SUBAPPLICATION Uebung_035a_AX (* Lauflicht 4 reine Zeitsteuerung (Adapter Version) *)
  (* Standard: 61499-2; Description: Copyright (c) 2026 Meisterschulen am Ostbahnhof This program and the accompanying materials are made available under the terms of the Eclipse Public License 2.0 which is available at https://www.eclipse.org/legal/epl-2.0/ SPDX-License-Identifier: EPL-2.0 *)
  (* Version 1.0, 2026-07-05, Franz Höpfinger, Meisterschulen am Ostbahnhof, generated solution *)
  PACKAGE Uebungen;
  IMPORT Uebungen::const::UT::DefaultPool::OutputNumber_N1;
  IMPORT logiBUS::io::DI::logiBUS_DI::Input_I1;
  IMPORT logiBUS::io::DI::logiBUS_DI::Input_I2;
  IMPORT logiBUS::io::DI::logiBUS_DI::Input_I3;
  IMPORT logiBUS::io::DI::logiBUS_DI::Input_I4;
  IMPORT logiBUS::io::DI::logiBUS_DI_Events::BUTTON_SINGLE_CLICK;
  IMPORT logiBUS::io::DQ::logiBUS_DO::Output_Q1;
  IMPORT logiBUS::io::DQ::logiBUS_DO::Output_Q2;
  IMPORT logiBUS::io::DQ::logiBUS_DO::Output_Q3;
  IMPORT logiBUS::io::DQ::logiBUS_DO::Output_Q4;
  IMPORT logiBUS::utils::sequence::const::sequence::NO_TIME;
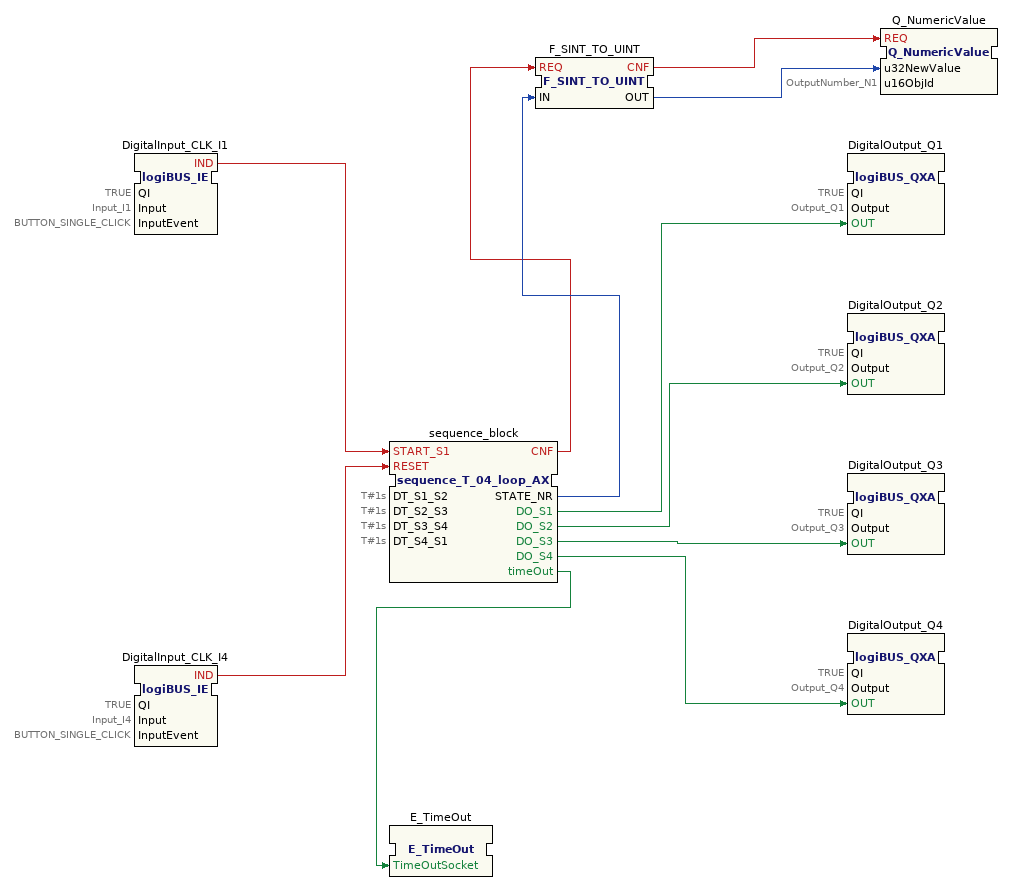
  FBS
    DigitalOutput_Q1 : logiBUS::io::DQ::logiBUS_QXA(QI := TRUE, Output := Output_Q1);
    DigitalOutput_Q2 : logiBUS::io::DQ::logiBUS_QXA(QI := TRUE, Output := Output_Q2);
    DigitalOutput_Q3 : logiBUS::io::DQ::logiBUS_QXA(QI := TRUE, Output := Output_Q3);
    DigitalOutput_Q4 : logiBUS::io::DQ::logiBUS_QXA(QI := TRUE, Output := Output_Q4);
    DigitalInput_CLK_I1 : logiBUS::io::DI::logiBUS_IE(QI := TRUE, Input := Input_I1, InputEvent := BUTTON_SINGLE_CLICK);
    DigitalInput_CLK_I4 : logiBUS::io::DI::logiBUS_IE(QI := TRUE, Input := Input_I4, InputEvent := BUTTON_SINGLE_CLICK);
    E_TimeOut : iec61499::events::E_TimeOut;
    Q_NumericValue : isobus::UT::Q::Q_NumericValue(u16ObjId := OutputNumber_N1);
    F_SINT_TO_UINT : iec61131::conversion::F_SINT_TO_UINT;
    sequence_block : logiBUS::utils::sequence::timed::sequence_T_04_loop_AX(DT_S1_S2 := T#1s, DT_S2_S3 := T#1s, DT_S3_S4 := T#1s, DT_S4_S1 := T#1s);
  END_FBS
  EVENT_CONNECTIONS
    F_SINT_TO_UINT.CNF TO Q_NumericValue.REQ;
    sequence_block.CNF TO F_SINT_TO_UINT.REQ;
    DigitalInput_CLK_I1.IND TO sequence_block.START_S1;
    DigitalInput_CLK_I4.IND TO sequence_block.RESET;
  END_CONNECTIONS
  DATA_CONNECTIONS
    F_SINT_TO_UINT.OUT TO Q_NumericValue.u32NewValue;
    sequence_block.STATE_NR TO F_SINT_TO_UINT.IN;
  END_CONNECTIONS
  ADAPTER_CONNECTIONS
    sequence_block.DO_S1 TO DigitalOutput_Q1.OUT;
    sequence_block.DO_S2 TO DigitalOutput_Q2.OUT;
    sequence_block.DO_S3 TO DigitalOutput_Q3.OUT;
    sequence_block.DO_S4 TO DigitalOutput_Q4.OUT;
    sequence_block.timeOut TO E_TimeOut.TimeOutSocket;
  END_CONNECTIONS
END_SUBAPPLICATION
